(*
Nazwa:			E_CapFeederState
Opis:			Stany sortera nasadek
Wersja:			v0.1
Data:			2022-07-13
Autor:			DP
Urzadzenia:		
Konfiguracja:	
Info:
*)


TYPE E_CapFeederState_1 :
(
	eDisabled:=0,			//Wyłączony
	eReady:=1,				//Gotowość
	eSleeveLowLevel:=2, 	//Praca, Niski poziom
	eSorting:=3,			//Praca
	eSleeveFull:=4			//Zapełniona
):=eDisabled;
END_TYPE

(* stored: Version 1.1.0.1, ProductVersion 3.1.4026.13, FileIdentifier dba2e3ede2a88fc71d43be19e5e10b8133ec23bf, FileSignature 30890741fd7bb6b92b9108c6e0da4b8c055bf8d1449d209b7bb6f1b161b386a278fd423883940e4efc27b53fd284c3be0b7dd762111d0f252978ce3f185e814d0a5f4801d292624a6cccd00e2909c93563cb3ed24862601b8487311e664f9cab62010c339a34c70dbed9c71162875a79ed839cdf032e89335cd93d47fa42e217c246dace4febc001537a731582c4247a3dd1b23f24ce4121db782a772d719e1f56001b535567fb17fb6dc589f2ab7b8653a333a8fa40e40b09c1a390045e4f7174c3d6cb8bfd4899e25c96f2ef306662751c910a01d2dc3772c18b5a0c9d7c8b76c371a40cb4a8223f0d6d2d1c47c036fa0c90b6c2d244e77663adc98bcc437b
   DUT E_CapFeederState_1: Id {65c5d9d6-8c28-4e29-aec7-7b6bee693dc0} *)
